FUNCTION_BLOCK COUNTER_HMI (* Service Interface Function Block Type *)
  (* Standard: 61499-2 *)
  (* Version 0.0, 2/4/2026, SESA713705, Schneider Electric, template *)
  PACKAGE SE.Nereda;
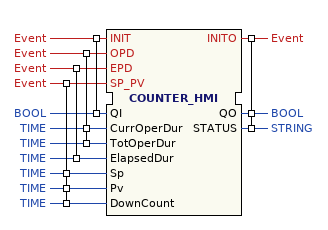
  EVENT_INPUT
    INIT WITH QI;
    OPD WITH CurrOperDur, TotOperDur;
    EPD WITH ElapsedDur;
    SP_PV WITH Sp, Pv, DownCount;
  END_EVENT
  EVENT_OUTPUT
    INITO WITH QO, STATUS;
  END_EVENT
  VAR_INPUT
    QI : BOOL;
    CurrOperDur : TIME;
    TotOperDur : TIME;
    ElapsedDur : TIME;
    Sp : TIME;
    Pv : TIME;
    DownCount : TIME;
  END_VAR
  VAR_OUTPUT
    QO : BOOL; (* Event Output Qualifier *)
    STATUS : STRING; (* Service Status *)
  END_VAR
  SERVICE /
    SEQUENCE 
    END_SEQUENCE
  END_SERVICE
END_FUNCTION_BLOCK
